(*udt (user defined type) of Beckhoff EL6900 - TwinSAFE Controller Status Interface:
	auth. Brent Lekx-Toniolo/Rob Remillard of Sodecia GTAC.; 
------------------------------------------------------------------------
REVISION NOTES:
	Version 1.0: November 2012
		- Initial Concept
	Version 20121204
		Changes from v1
			- Change to Naming Convention to include date as version
	Version 20150925
			- Added variable for area to store terminal temperature data, b.lekx-toniolo
			- Changed InfoData to EX type to allow linking area for AMS and Port, b.lekx-toniolo
	Version 20160426
			- Added Instance of udt_EL6900_DeviceInfoData_yyyymmdd, b.lekx-toniolo

------------------------------------------------------------------------

*)

TYPE udt_EP1918_STAT_20250213 :
	STRUCT
	SGs_FB_ERR: BYTE;
	(*
	FB ERROR Status Summary of ALL FBs in Terminal, 1 bit per SG*)

	SGs_COM_ERR: BYTE;
	(*
	COM Status of all Coms Linked to Terminal, 1 bit per SG*)

	SGs_OUT_ERR: BYTE;
	(*
	OUTPUT ERROR Status of all Outputs Linked to Terminal, 1 bit per SG*)

	FBs_FB_ERR: DINT;
	(*
	FB ERROR Status fof EACH FB within Terminal, 1 bit per FB*)

	I: BYTE;

	Device_Info_Data: udt_EL6900_DeviceInfoData_20160426;
	InfoData: udt_ECATSlave_StatusEXT;

	(*CoE Data Section*)
	CoE_Project_State:	UDINT;	(*Retreived via CoE - For Storage of Safety Project State*)
	CoE_Temperature_1: 	UINT; 	(*Retreived via CoE - For Storage of Primary Temperature MC1 Data*)
	CoE_Temperature_2: 	UINT;  	(*Retreived via CoE - For Storage of Secondary Temperature MC1 Data*)


	END_STRUCT
END_TYPE

(* stored: Version 1.1.0.1, ProductVersion 3.1.4024.12
   DUT udt_EP1918_STAT_20250213: Id {a63e92a9-64c8-43b7-942d-5ee219272f3c} *)
